(* IEC 61131-3 sources: mect_apps/TPAC1008/RemoteControl_PLC, 7 files *)

(* ---- ImpostazioniCAN1.gvl ---- *)
(* Global var file *)
VAR_GLOBAL
	ch1_CAN1_IN_DIG_8_1 AT %IB3.4096: BYTE;
	ch1_CAN1_IN_DIG_8_2 AT %IB3.4097: BYTE;
	ch1_CAN1_OUT_DIG_8_1 AT %QB3.4096: BYTE;

	ch1_CAN1_OUT_DIG_8_1_7 AT %QX3.4096.7: BOOL;

	ch1_CAN1_OUT_DIG_8_2 AT %QB3.4097: BYTE;
	ch1_CAN1_IN_AN_1 AT %IW3.8192: INT;
	ch1_CAN1_IN_AN_2 AT %IW3.8194: INT;
	ch1_CAN1_IN_AN_3 AT %IW3.8196: INT;
	ch1_CAN1_IN_AN_4 AT %IW3.8198: INT;
	ch1_CAN1_IN_AN_5 AT %IW3.8200: INT;
	ch1_CAN1_IN_AN_6 AT %IW3.8202: INT;
	ch1_CAN1_IN_AN_7 AT %IW3.8204: INT;
	ch1_CAN1_IN_AN_8 AT %IW3.8206: INT;
	ch1_CAN1_IN_AN_9 AT %IW3.8208: INT;
	ch1_CAN1_IN_AN_10 AT %IW3.8210: INT;
	ch1_CAN1_IN_AN_11 AT %IW3.8212: INT;
	ch1_CAN1_IN_AN_12 AT %IW3.8214: INT;
	ch1_CAN1_IN_AN_13 AT %IW3.8216: INT;
	ch1_CAN1_IN_AN_14 AT %IW3.8218: INT;
	ch1_CAN1_IN_AN_15 AT %IW3.8220: INT;
	ch1_CAN1_IN_AN_16 AT %IW3.8222: INT;
	ch1_CAN1_OUT_AN_1 AT %QW3.8192: INT;
	PLC_CAN1_IN_DIG_8_1 AT %MB0.21200: BYTE;

	PLC_CAN1_IN_DIG_8_2 AT %MB0.21204: BYTE;
	PLC_CAN1_OUT_DIG_8_1 AT %MB0.21208: BYTE;
	PLC_CAN1_OUT_DIG_8_1_0 AT %MX0.21208.0: BOOL;
	PLC_CAN1_OUT_DIG_8_1_1 AT %MX0.21208.1: BOOL;
	PLC_CAN1_OUT_DIG_8_1_2 AT %MX0.21208.2: BOOL;
	PLC_CAN1_OUT_DIG_8_1_3 AT %MX0.21208.3: BOOL;
	PLC_CAN1_OUT_DIG_8_1_4 AT %MX0.21208.4: BOOL;
	PLC_CAN1_OUT_DIG_8_1_5 AT %MX0.21208.5: BOOL;
	PLC_CAN1_OUT_DIG_8_1_6 AT %MX0.21208.6: BOOL;
	PLC_CAN1_OUT_DIG_8_1_7 AT %MX0.21208.7: BOOL;

	PLC_CAN1_OUT_DIG_8_2 AT %MB0.21212: BYTE;

	PLC_CAN1_IN_AN_1 AT %MW0.21216: INT;
	PLC_CAN1_IN_AN_2 AT %MW0.21220: INT;
	PLC_CAN1_IN_AN_3 AT %MW0.21224: INT;
	PLC_CAN1_IN_AN_4 AT %MW0.21228: INT;
	PLC_CAN1_IN_AN_5 AT %MW0.21232: INT;
	PLC_CAN1_IN_AN_6 AT %MW0.21236: INT;
	PLC_CAN1_IN_AN_7 AT %MW0.21240: INT;
	PLC_CAN1_IN_AN_8 AT %MW0.21244: INT;
	PLC_CAN1_IN_AN_9 AT %MW0.21248: INT;
	PLC_CAN1_IN_AN_10 AT %MW0.21252: INT;
	PLC_CAN1_IN_AN_11 AT %MW0.21256: INT;
	PLC_CAN1_IN_AN_12 AT %MW0.21260: INT;
	PLC_CAN1_IN_AN_13 AT %MW0.21264: INT;
	PLC_CAN1_IN_AN_14 AT %MW0.21268: INT;
	PLC_CAN1_IN_AN_15 AT %MW0.21272: INT;
	PLC_CAN1_IN_AN_16 AT %MW0.21276: INT;
	PLC_CAN1_OUT_AN_1 AT %MW0.21280: INT;
END_VAR

(* ---- Resource1.gvl ---- *)
(* Global variable file *)
VAR_GLOBAL

	Selection AT %MW0.4:UINT;
	ISI_S1_GRU AT %MW0.8:INT;
	FSI_S1_GRU AT %MW0.12:INT;
	ISL_S1_GRU AT %MW0.16:INT;
	FSL_S1_GRU AT %MW0.20:INT;
	ISI_S2_GRU AT %MW0.24:INT;
	FSI_S2_GRU AT %MW0.28:INT;
	ISL_S2_GRU AT %MW0.32:INT;
	FSL_S2_GRU AT %MW0.36:INT;
	ISI_S3_GRU AT %MW0.40:INT;
	FSI_S3_GRU AT %MW0.44:INT;
	ISL_S3_GRU AT %MW0.48:INT;
	FSL_S3_GRU AT %MW0.52:INT;
	ISI_S1_ESC AT %MW0.56:INT;
	FSI_S1_ESC AT %MW0.60:INT;
	ISL_S1_ESC AT %MW0.64:INT;
	FSL_S1_ESC AT %MW0.68:INT;
	ISI_S2_ESC AT %MW0.72:INT;
	FSI_S2_ESC AT %MW0.76:INT;
	ISL_S2_ESC AT %MW0.80:INT;
	FSL_S2_ESC AT %MW0.84:INT;
	ISI_S3_ESC AT %MW0.88:INT;
	FSI_S3_ESC AT %MW0.92:INT;
	ISL_S3_ESC AT %MW0.96:INT;
	FSL_S3_ESC AT %MW0.100:INT;
	ZERO_S1_GRU AT %MW0.104:INT;
	ZERO_S2_GRU AT %MW0.108:INT;
	ZERO_S3_GRU AT %MW0.112:INT;
	ZERO_S1_ESC AT %MW0.116:INT;
	ZERO_S2_ESC AT %MW0.120:INT;
	ZERO_S3_ESC AT %MW0.124:INT;
	manual AT %MW0.128:UINT;
	DigitalOutput_1 AT %MD0.5380:UDINT;
	DigitalOutput_2 AT %MD0.5384:UDINT;
	DigitalInput_3 AT %MD0.5388:UDINT;
	DigitalInput_4 AT %MD0.5392:UDINT;
	TimeValue AT %MD0.5396:REAL;
	TimeMin AT %MD0.5400:REAL;
	TimeMax AT %MD0.5404:REAL;
	AnalogInput_1 AT %MW0.5408:INT;
	AnalogInput_2 AT %MW0.5412:INT;
	Mesaure_gru1 AT %MW0.5416:INT;
	Mesaure_gru2 AT %MW0.5420:INT;
	Mesaure_gru3 AT %MW0.5424:INT;
	Mesaure_esc1 AT %MW0.5428:INT;
	Mesaure_esc2 AT %MW0.5432:INT;
	Mesaure_esc3 AT %MW0.5436:INT;
	Tasto1 AT %MW0.5440:INT;
	Tasto2 AT %MW0.5444:INT;
	Tasto3 AT %MW0.5448:INT;
	Tasto4 AT %MW0.5452:INT;
	Tasto5 AT %MW0.5456:INT;
	Tasto6 AT %MW0.5460:INT;

	step1T AT %MW0.5464:INT;
	step1M AT %MW0.5468:INT;
	step2T AT %MW0.5472:INT;
	step2M AT %MW0.5476:INT;
	step3T AT %MW0.5480:INT;
	step3M AT %MW0.5484:INT;
	step4T AT %MW0.5488:INT;
	step4M AT %MW0.5492:INT;
	step5T AT %MW0.5496:INT;
	step5M AT %MW0.5500:INT;
	step6T AT %MW0.5504:INT;
	step6M AT %MW0.5508:INT;
	step7T AT %MW0.5512:INT;
	step7M AT %MW0.5516:INT;
	step8T AT %MW0.5520:INT;
	step8M AT %MW0.5524:INT;
	step9T AT %MW0.5528:INT;
	step9M AT %MW0.5532:INT;
	step10T AT %MW0.5536:INT;
	step10M AT %MW0.5540:INT;
	SetZ_gru1 AT %MW0.5544:INT;
	SetZ_gru2 AT %MW0.5548:INT;
	SetZ_gru3 AT %MW0.5552:INT;
	SetZ_esc1 AT %MW0.5556:INT;
	SetZ_esc2 AT %MW0.5560:INT;
	SetZ_esc3 AT %MW0.5564:INT;

	Offset_AnIn_1_GRU:INT;
	Offset_AnIn_2_GRU:INT;
	Offset_AnIn_3_GRU:INT;
	Offset_AnIn_1_ESC:INT;
	Offset_AnIn_2_ESC:INT;
	Offset_AnIn_3_ESC:INT;

END_VAR

(* ---- TPACLocaIO.gvl ---- *)
(*Global variable file*)
(*[[
]]*)
VAR_GLOBAL
	PLC_DigIn_1 AT %MW0.21200:WORD;
	PLC_DigIn_2 AT %MW0.21204:WORD;
	PLC_DigIn_3 AT %MW0.21208:WORD;
	PLC_DigIn_4 AT %MW0.21212:WORD;
	PLC_DigIn_5 AT %MW0.21216:WORD;
	PLC_DigIn_6 AT %MW0.21220:WORD;
	PLC_DigIn_7 AT %MW0.21224:WORD;
	PLC_DigIn_8 AT %MW0.21228:WORD;
	PLC_DigIn_9 AT %MW0.21232:WORD;
	PLC_DigIn_10 AT %MW0.21236:WORD;
	PLC_DigIn_11 AT %MW0.21240:WORD;
	PLC_DigIn_12 AT %MW0.21244:WORD;
	PLC_DigIn_13 AT %MW0.21248:WORD;
	PLC_DigIn_14 AT %MW0.21252:WORD;
	PLC_DigIn_15 AT %MW0.21256:WORD;
	PLC_DigIn_16 AT %MW0.21260:WORD;
	PLC_DigOut_1 AT %MW0.21264:WORD;
	PLC_DigOut_2 AT %MW0.21268:WORD;
	PLC_DigOut_3 AT %MW0.21272:WORD;
	PLC_DigOut_4 AT %MW0.21276:WORD;
	PLC_DigOut_5 AT %MW0.21280:WORD;
	PLC_DigOut_6 AT %MW0.21284:WORD;
	PLC_DigOut_7 AT %MW0.21288:WORD;
	PLC_DigOut_8 AT %MW0.21292:WORD;
	PLC_DigOut_9 AT %MW0.21296:WORD;
	PLC_DigOut_10 AT %MW0.21300:WORD;
	PLC_DigOut_11 AT %MW0.21304:WORD;
	PLC_DigOut_12 AT %MW0.21308:WORD;
	PLC_DigOut_13 AT %MW0.21312:WORD;
	PLC_DigOut_14 AT %MW0.21316:WORD;
	PLC_DigOut_15 AT %MW0.21320:WORD;
	PLC_DigOut_16 AT %MW0.21324:WORD;
	PLC_DigDir_1 AT %MW0.21328:WORD;
	PLC_DigDir_2 AT %MW0.21332:WORD;
	PLC_DigDir_3 AT %MW0.21336:WORD;
	PLC_DigDir_4 AT %MW0.21340:WORD;
	PLC_DigDir_5 AT %MW0.21344:WORD;
	PLC_DigDir_6 AT %MW0.21348:WORD;
	PLC_DigDir_7 AT %MW0.21352:WORD;
	PLC_DigDir_8 AT %MW0.21356:WORD;
	PLC_DigDir_9 AT %MW0.21360:WORD;
	PLC_DigDir_10 AT %MW0.21364:WORD;
	PLC_DigDir_11 AT %MW0.21368:WORD;
	PLC_DigDir_12 AT %MW0.21372:WORD;
	PLC_DigDir_13 AT %MW0.21376:WORD;
	PLC_DigDir_14 AT %MW0.21380:WORD;
	PLC_DigDir_15 AT %MW0.21384:WORD;
	PLC_DigDir_16 AT %MW0.21388:WORD;
	PLC_AnIn_1 AT %MW0.21392:INT;
	PLC_AnIn_2 AT %MW0.21396:INT;
	PLC_AnIn_3 AT %MW0.21400:INT;
	PLC_AnIn_4 AT %MW0.21404:INT;
	PLC_AnIn_5 AT %MW0.21408:INT;
	PLC_AnIn_6 AT %MW0.21412:INT;
	PLC_AnIn_7 AT %MW0.21416:INT;
	PLC_AnIn_8 AT %MW0.21420:INT;
	PLC_AnOut_1  AT %MW0.21424:INT;
	PLC_AnOut_2 AT %MW0.21428:INT;
	PLC_AnOut_3  AT %MW0.21432:INT;
	PLC_AnOut_4 AT %MW0.21436:INT;
	PLC_AnOut_5  AT %MW0.21440:INT;
	PLC_AnOut_6 AT %MW0.21444:INT;
	PLC_AnOut_7  AT %MW0.21448:INT;
	PLC_AnOut_8 AT %MW0.21452:INT;
	PLC_AnInConf_1 AT %MW0.21456:WORD;
	PLC_AnInConf_2 AT %MW0.21460:WORD;
	PLC_AnInConf_3 AT %MW0.21464:WORD;
	PLC_AnInConf_4 AT %MW0.21468:WORD;
	PLC_AnInConf_5 AT %MW0.21472:WORD;
	PLC_AnInConf_6 AT %MW0.21476:WORD;
	PLC_AnInConf_7 AT %MW0.21480:WORD;
	PLC_AnInConf_8 AT %MW0.21484:WORD;
	PLC_AnOutConf_1 AT %MW0.21488:WORD;
	PLC_AnOutConf_2 AT %MW0.21492:WORD;
	PLC_AnOutConf_3 AT %MW0.21496:WORD;
	PLC_AnOutConf_4 AT %MW0.21500:WORD;
	PLC_AnOutConf_5 AT %MW0.21504:WORD;
	PLC_AnOutConf_6 AT %MW0.21508:WORD;
	PLC_AnOutConf_7 AT %MW0.21512:WORD;
	PLC_AnOutConf_8 AT %MW0.21516:WORD;
	PLC_Tamb AT %MW0.21520:INT;
	PLC_EncoderLo AT %MW0.21524:UINT;
	PLC_EncoderHi AT %MW0.21528:UINT;
	PLC_StatusReg AT %MW0.21532:UINT;
	PLC_ControlWord  AT %MW0.21536:WORD;
	PLC_EncoderPreset_Lo AT %MW0.21540:UINT;
	PLC_EncoderPreset_Hi AT %MW0.21544:UINT;
	PLC_EncoderReset AT %MW0.21548:WORD;
	PLC_EncoderEnable AT %MW0.21552:WORD;
	PLC_RPM AT %MW0.21556:UINT;
	PLC_time AT %MD0.21560:REAL;
	PLC_timeMin AT %MD0.21564:REAL;
	PLC_timeMax AT %MD0.21568:REAL;
END_VAR

(* ---- fb_TPAC1006_LIOsync.st ---- *)
(*[[
]]*)
FUNCTION_BLOCK fb_TPAC1006_LIOsync
#import "LIO_TPAC1006.gvl"
#import "TPACLocaIO.gvl"
#import "crosstable.gvl"
VAR_INPUT
END_VAR
VAR
END_VAR
IF (HardwareType AND 16#000000FF) >= 16#1 THEN
	IF (UINT_TO_WORD(TP1006_LIO_StatusReg) AND 16#01) = 1 	 THEN

		PLC_DigIn_1:=BOOL_TO_WORD(TP1006_LIO_DigIn_1);
		PLC_DigIn_2:=BOOL_TO_WORD(TP1006_LIO_DigIn_2);
		PLC_DigIn_3:=BOOL_TO_WORD(TP1006_LIO_DigIn_3);
		PLC_DigIn_4:=BOOL_TO_WORD(TP1006_LIO_DigIn_4);
		PLC_DigIn_5:=BOOL_TO_WORD(TP1006_LIO_DigIn_5);
		PLC_DigIn_6:=BOOL_TO_WORD(TP1006_LIO_DigIn_6);
		PLC_DigIn_7:=BOOL_TO_WORD(TP1006_LIO_DigIn_7);
		PLC_DigIn_8:=BOOL_TO_WORD(TP1006_LIO_DigIn_8);

		PLC_DigIn_9:=BOOL_TO_WORD(TP1006_LIO_DigIn_9);
		PLC_DigIn_10:=BOOL_TO_WORD(TP1006_LIO_DigIn_10);
		PLC_DigIn_11:=BOOL_TO_WORD(TP1006_LIO_DigIn_11);
		PLC_DigIn_12:=BOOL_TO_WORD(TP1006_LIO_DigIn_12);
		PLC_DigIn_13:=BOOL_TO_WORD(TP1006_LIO_DigIn_13);
		PLC_DigIn_14:=BOOL_TO_WORD(TP1006_LIO_DigIn_14);
		PLC_DigIn_15:=BOOL_TO_WORD(TP1006_LIO_DigIn_15);
		PLC_DigIn_16:=BOOL_TO_WORD(TP1006_LIO_DigIn_16);

		TP1006_LIO_DigOut_1:=WORD_TO_BOOL(PLC_DigOut_1);
		TP1006_LIO_DigOut_2:=WORD_TO_BOOL(PLC_DigOut_2);
		TP1006_LIO_DigOut_3:=WORD_TO_BOOL(PLC_DigOut_3);
		TP1006_LIO_DigOut_4:=WORD_TO_BOOL(PLC_DigOut_4);
		TP1006_LIO_DigOut_5:=WORD_TO_BOOL(PLC_DigOut_5);
		TP1006_LIO_DigOut_6:=WORD_TO_BOOL(PLC_DigOut_6);
		TP1006_LIO_DigOut_7:=WORD_TO_BOOL(PLC_DigOut_7);
		TP1006_LIO_DigOut_8:=WORD_TO_BOOL(PLC_DigOut_8);

		TP1006_LIO_DigOut_9:=WORD_TO_BOOL(PLC_DigOut_9);
		TP1006_LIO_DigOut_10:=WORD_TO_BOOL(PLC_DigOut_10);
		TP1006_LIO_DigOut_11:=WORD_TO_BOOL(PLC_DigOut_11);
		TP1006_LIO_DigOut_12:=WORD_TO_BOOL(PLC_DigOut_12);
		TP1006_LIO_DigOut_13:=WORD_TO_BOOL(PLC_DigOut_13);
		TP1006_LIO_DigOut_14:=WORD_TO_BOOL(PLC_DigOut_14);
		TP1006_LIO_DigOut_15:=WORD_TO_BOOL(PLC_DigOut_15);
		TP1006_LIO_DigOut_16:=WORD_TO_BOOL(PLC_DigOut_16);

		PLC_AnIn_1:= TP1006_LIO_AnIn_1;
		PLC_AnIn_2:= TP1006_LIO_AnIn_2;
		PLC_AnIn_3:= TP1006_LIO_AnIn_3;
		PLC_AnIn_4:= TP1006_LIO_AnIn_4;

		PLC_Tamb:= TP1006_LIO_Tamb;
		PLC_EncoderLo:= TP1006_LIO_EncoderLo;
		PLC_EncoderHi:= TP1006_LIO_EncoderHi;
		PLC_StatusReg:= TP1006_LIO_StatusReg;
		PLC_RPM:= TP1006_LIO_RPM;
		TP1006_LIO_AnIn_Conf:=WORD_TO_INT(PLC_AnInConf_1 OR SHL(PLC_AnInConf_2,4) OR SHL(PLC_AnInConf_3,8) OR SHL(PLC_AnInConf_4,12) );
		TP1006_LIO_AnOut_Conf:=WORD_TO_INT(INT_TO_WORD(WORD_TO_INT(PLC_AnOutConf_1)) OR SHL(INT_TO_WORD(WORD_TO_INT(PLC_AnOutConf_2)),4) );

		TP1006_LIO_AnOut_1:= PLC_AnOut_1;
		TP1006_LIO_AnOut_2:= PLC_AnOut_2;
		TP1006_LIO_ControlWord:= PLC_ControlWord;
		TP1006_LIO_EncoderPreset_Lo:= PLC_EncoderPreset_Lo;
		TP1006_LIO_EncoderPreset_hI:= PLC_EncoderPreset_Hi;
	END_IF;

END_IF;

END_FUNCTION_BLOCK

(* ---- fb_TPAC1007_LIOsync.st ---- *)
(*[[
]]*)
FUNCTION_BLOCK fb_TPAC1007_LIOsync
#import "LIO_TPAC1007.gvl"
#import "TPACLocaIO.gvl"
#import "crosstable.gvl"
VAR_INPUT
END_VAR
VAR
	tmp_dig_out: BYTE;
	tmp_dig_outold:BYTE;
	tmp_dig_dir: BYTE;
	tmp_dig_dirold:BYTE;
END_VAR

IF (HardwareType AND 16#00FF0000) >= 16#1 THEN
		PLC_StatusReg:=TP1007_LIO_Revision;
		PLC_DigIn_1:=BOOL_TO_WORD(TP1007_LIO_DigIn_1);
		PLC_DigIn_2:=BOOL_TO_WORD(TP1007_LIO_DigIn_2);
		PLC_DigIn_3:=BOOL_TO_WORD(TP1007_LIO_DigIn_3);
		PLC_DigIn_4:=BOOL_TO_WORD(TP1007_LIO_DigIn_4);
		PLC_DigIn_5:=BOOL_TO_WORD(TP1007_LIO_DigIn_5);
		PLC_DigIn_6:=BOOL_TO_WORD(TP1007_LIO_DigIn_6);
		PLC_DigIn_7:=BOOL_TO_WORD(TP1007_LIO_DigIn_7);
		PLC_DigIn_8:=BOOL_TO_WORD(TP1007_LIO_DigIn_8);
		PLC_DigIn_9:=BOOL_TO_WORD(TP1007_LIO_DigIn_9);
		PLC_DigIn_10:=BOOL_TO_WORD(TP1007_LIO_DigIn_10);
		PLC_DigIn_11:=BOOL_TO_WORD(TP1007_LIO_DigIn_11);
		PLC_DigIn_12:=BOOL_TO_WORD(TP1007_LIO_DigIn_12);

		PLC_Tamb:= TP1007_LIO_Tamb;
		PLC_EncoderLo:= TP1007_LIO_EncoderLo;
		PLC_EncoderHi:= TP1007_LIO_EncoderHi;

		PLC_AnIn_1 := TP1007_LIO_AnIn_1;
		PLC_AnIn_2 := TP1007_LIO_AnIn_2;

(*SCRITTURA 1*)
		tmp_dig_dir := WORD_TO_BYTE(PLC_DigDir_1 OR SHL(PLC_DigDir_2,1) OR SHL(PLC_DigDir_3,2) OR SHL(PLC_DigDir_4,3) OR SHL(PLC_DigDir_5,4) OR SHL(PLC_DigDir_6,5) OR SHL(PLC_DigDir_7,6) OR SHL(PLC_DigDir_8,7) );
		IF tmp_dig_dir <> tmp_dig_dirold THEN
			TP1007_LIO_DigDir_1_8 := tmp_dig_dir;
		END_IF;
		tmp_dig_dirold := tmp_dig_dir;

(*SCRITTURA 2*)
		tmp_dig_out:= WORD_TO_BYTE(PLC_DigOut_1 OR SHL(PLC_DigOut_2,1) OR SHL(PLC_DigOut_3,2) OR SHL(PLC_DigOut_4,3) OR SHL(PLC_DigOut_5,4) OR SHL(PLC_DigOut_6,5) OR SHL(PLC_DigOut_7,6) OR SHL(PLC_DigOut_8,7) );
		IF tmp_dig_out<> tmp_dig_outold THEN
			TP1007_LIO_DigOut_1_8:= tmp_dig_out;
		END_IF;
		tmp_dig_outold:=tmp_dig_out;

(*SCRITTURA 3*)
		IF PLC_AnInConf_1 <> TP1007_LIO_AnInConf_1 THEN
			TP1007_LIO_AnInConf_1 := PLC_AnInConf_1 ;
		END_IF;
(*SCRITTURA 4*)
		IF PLC_AnInConf_2 <> TP1007_LIO_AnInConf_2 THEN
			TP1007_LIO_AnInConf_2 := PLC_AnInConf_2 ;
		END_IF;
(*SCRITTURA 5*)
		IF PLC_AnOutConf_1 <> TP1007_LIO_AnOut_Conf THEN
			TP1007_LIO_AnOut_Conf := PLC_AnOutConf_1;
		END_IF;
(*SCRITTURA 6*)
		IF PLC_AnOut_1 <> (TP1007_LIO_AnOut_1) THEN
			TP1007_LIO_AnOut_1 := PLC_AnOut_1;
		END_IF;
(*SCRITTURA 7*)
		IF PLC_EncoderReset <> TP1007_LIO_EncoderReset THEN
			TP1007_LIO_EncoderReset := PLC_EncoderReset;
		END_IF;
(*SCRITTURA 8*)
		IF PLC_EncoderEnable <> TP1007_LIO_EncoderEnable THEN
			TP1007_LIO_EncoderEnable := PLC_EncoderEnable;
		END_IF;

END_IF;
END_FUNCTION_BLOCK

(* ---- PLC.st ---- *)
(*[[
]]*)
PROGRAM PLC
#import "crosstable.gvl"
#import "Resource1.gvl"
#import "LIO_TPAC1006.gvl"
#import "TPACLocaIO.gvl"
VAR
	FIRST_CYCLE:BOOL;
	LAST_BUTTON :UINT;
	TMP1:REAL;
	TMP2:REAL;
END_VAR;
	IF NOT FIRST_CYCLE THEN
		IF Selection > 0 THEN
(*
			ISI_S1_GRU:=4000;
			FSI_S1_GRU:=20000;
			ISI_S2_GRU:=4000;
			FSI_S2_GRU:=20000;
			ISI_S3_GRU:=4000;
			FSI_S3_GRU:=20000;
			ISI_S1_ESC:=4000;
			FSI_S1_ESC:=20000;
			ISI_S2_ESC:=4000;
			FSI_S2_ESC:=20000;
			ISI_S3_ESC:=4000;
			FSI_S3_ESC:=20000;

			ISL_S1_GRU:=0;
			FSL_S1_GRU:=3600;
			ISL_S2_GRU:=0;
			FSL_S2_GRU:=3600;
			ISL_S3_GRU:=-900;
			FSL_S3_GRU:=900;
			ISL_S1_ESC:=0;
			FSL_S1_ESC:=3000;
			ISL_S2_ESC:=0;
			FSL_S2_ESC:=3600;
			ISL_S3_ESC:=-900;
			FSL_S3_ESC:=900;
	*)
			FIRST_CYCLE:=TRUE;
		END_IF;
	ELSE
		IF Selection =1 THEN
			PLC_AnInConf_1:=1;
			PLC_AnInConf_2:=1;
			PLC_AnInConf_3:=2;
			PLC_AnInConf_4:=0;
		ELSE
			PLC_AnInConf_1:=1;
			PLC_AnInConf_2:=1;
			PLC_AnInConf_3:=1;
			PLC_AnInConf_4:=0;
		END_IF;
		IF SetZ_gru1 =1 THEN
			ZERO_S1_GRU:=PLC_AnIn_1;
		END_IF;

		IF SetZ_gru2 = 1 THEN
			ZERO_S2_GRU:=PLC_AnIn_2;
		END_IF;

		IF SetZ_gru3 = 1 THEN
			ZERO_S3_GRU:=PLC_AnIn_3;
		END_IF;

		IF SetZ_esc1  = 1 THEN
			ZERO_S1_ESC:=PLC_AnIn_1;
		END_IF;

		IF SetZ_esc2  = 1 THEN
			ZERO_S2_ESC:=PLC_AnIn_2;
		END_IF;

		IF SetZ_esc3  = 1 THEN
			ZERO_S3_ESC:=PLC_AnIn_3;
		END_IF;

		IF Selection = 2 THEN
			IF Tasto1 =1 THEN
				IF LAST_BUTTON <> 1 THEN
					PLC_DigOut_1:=0;
					PLC_DigOut_2:=0;
					LAST_BUTTON:=1;
				ELSE
					PLC_DigOut_1:=1;
					PLC_DigOut_2:=0;
					PLC_DigOut_3:=0;
				END_IF;
			ELSIF Tasto2 =1 THEN
				IF LAST_BUTTON <> 2 THEN
					PLC_DigOut_1:=0;
					PLC_DigOut_2:=0;
					LAST_BUTTON:=2;
				ELSE
					PLC_DigOut_1:=0;
					PLC_DigOut_2:=1;
					PLC_DigOut_3:=1;
				END_IF;
			ELSIF Tasto3 =1 THEN
				IF LAST_BUTTON <> 3 THEN
					PLC_DigOut_4:=0;
					PLC_DigOut_5:=0;
					LAST_BUTTON:=3;
				ELSE
					PLC_DigOut_4:=1;
					PLC_DigOut_5:=0;
					PLC_DigOut_6:=0;
				END_IF;
			ELSIF Tasto4 =1 THEN
				IF LAST_BUTTON <> 4 THEN
					PLC_DigOut_4:=0;
					PLC_DigOut_5:=0;
					LAST_BUTTON:=4;
				ELSE
					PLC_DigOut_4:=0;
					PLC_DigOut_5:=1;
					PLC_DigOut_6:=1;
				END_IF;
			ELSIF Tasto5 =1 THEN
				IF LAST_BUTTON <> 5 THEN
					PLC_DigOut_7:=0;
					PLC_DigOut_8:=0;
					LAST_BUTTON:=5;
				ELSE
					PLC_DigOut_7:=1;
					PLC_DigOut_8:=0;
					PLC_DigOut_9:=0;
				END_IF;
			ELSIF Tasto6 =1 THEN
				IF LAST_BUTTON <> 6 THEN
					PLC_DigOut_7:=0;
					PLC_DigOut_8:=0;
					LAST_BUTTON:=6;
				ELSE
					PLC_DigOut_7:=0;
					PLC_DigOut_8:=1;
					PLC_DigOut_9:=1;
				END_IF;
			ELSIF Tasto1=0 AND Tasto2=0 AND Tasto3=0 AND Tasto4=0 AND Tasto5=0 AND Tasto6=0 THEN
				PLC_DigOut_1:=0;
				PLC_DigOut_2:=0;
				PLC_DigOut_4:=0;
				PLC_DigOut_5:=0;
				PLC_DigOut_7:=0;
				PLC_DigOut_8:=0;
			END_IF;

			IF(FSI_S1_ESC-ISI_S1_ESC) > 0 THEN
				TMP1:=INT_TO_REAL((ZERO_S1_ESC-ISI_S1_ESC))*int_to_real((FSL_S1_ESC-ISL_S1_ESC))/INT_TO_REAL((FSI_S1_ESC-ISI_S1_ESC))+INT_TO_REAL(ISL_S1_ESC);
				TMP2:=INT_TO_REAL((PLC_AnIn_1-ISI_S1_ESC))*int_to_real((FSL_S1_ESC-ISL_S1_ESC))/INT_TO_REAL((FSI_S1_ESC-ISI_S1_ESC))+INT_TO_REAL(ISL_S1_ESC);
				Mesaure_ESC1:=REAL_TO_INT(TMP2-TMP1);
			END_IF;
			IF(FSI_S2_ESC-ISI_S2_ESC) > 0 THEN
				TMP1:=INT_TO_REAL((ZERO_S2_ESC-ISI_S2_ESC))*int_to_real((FSL_S2_ESC-ISL_S2_ESC))/INT_TO_REAL((FSI_S2_ESC-ISI_S2_ESC))+INT_TO_REAL(ISL_S2_ESC);
				TMP2:=INT_TO_REAL((PLC_AnIn_2-ISI_S2_ESC))*int_to_real((FSL_S2_ESC-ISL_S2_ESC))/INT_TO_REAL((FSI_S2_ESC-ISI_S2_ESC))+INT_TO_REAL(ISL_S2_ESC);
				Mesaure_ESC2:=REAL_TO_INT(TMP2-TMP1);
			END_IF;
			IF(FSI_S3_ESC-ISI_S3_ESC) > 0 THEN
				TMP1:=INT_TO_REAL((ZERO_S3_ESC-ISI_S3_ESC))*int_to_real((FSL_S3_ESC-ISL_S3_ESC))/INT_TO_REAL((FSI_S3_ESC-ISI_S3_ESC))+INT_TO_REAL(ISL_S3_ESC);
				TMP2:=INT_TO_REAL((PLC_AnIn_3-ISI_S3_ESC))*int_to_real((FSL_S3_ESC-ISL_S3_ESC))/INT_TO_REAL((FSI_S3_ESC-ISI_S3_ESC))+INT_TO_REAL(ISL_S3_ESC);
				Mesaure_ESC3:=REAL_TO_INT(TMP2-TMP1);

			END_IF;

		ELSIF Selection = 1 THEN
			IF Tasto1 =1 THEN
				IF LAST_BUTTON <> 1 THEN
					PLC_DigOut_1:=0;
					PLC_DigOut_2:=0;
					LAST_BUTTON:=1;
				ELSE
					PLC_DigOut_1:=1;
					PLC_DigOut_2:=0;
				END_IF;
			ELSIF Tasto2 =1 THEN
				IF LAST_BUTTON <> 2 THEN
					PLC_DigOut_1:=0;
					PLC_DigOut_2:=0;
					LAST_BUTTON:=2;
				ELSE
					PLC_DigOut_1:=0;
					PLC_DigOut_2:=1;
				END_IF;
			ELSIF Tasto3 =1 THEN
				IF LAST_BUTTON <> 3 THEN
					PLC_DigOut_3:=0;
					PLC_DigOut_4:=0;
					LAST_BUTTON:=3;
				ELSE
					PLC_DigOut_3:=1;
					PLC_DigOut_4:=0;
				END_IF;
			ELSIF Tasto4 =1 THEN
				IF LAST_BUTTON <> 4 THEN
					PLC_DigOut_3:=0;
					PLC_DigOut_4:=0;
					LAST_BUTTON:=4;
				ELSE
					PLC_DigOut_3:=0;
					PLC_DigOut_4:=1;
				END_IF;
			ELSIF Tasto1=0 AND Tasto2=0 AND Tasto3=0 AND Tasto4=0 AND Tasto5=0 AND Tasto6=0 THEN
				PLC_DigOut_1:=0;
				PLC_DigOut_2:=0;
				PLC_DigOut_3:=0;
				PLC_DigOut_4:=0;
				PLC_DigOut_7:=0;
				PLC_DigOut_8:=0;
			END_IF;

			IF(FSI_S1_GRU-ISI_S1_GRU) > 0 THEN
				TMP1:=INT_TO_REAL((ZERO_S1_GRU-ISI_S1_GRU))*int_to_real((FSL_S1_GRU-ISL_S1_GRU))/INT_TO_REAL((FSI_S1_GRU-ISI_S1_GRU))+INT_TO_REAL(ISL_S1_GRU);
				TMP2:=INT_TO_REAL((PLC_AnIn_1-ISI_S1_GRU))*int_to_real((FSL_S1_GRU-ISL_S1_GRU))/INT_TO_REAL((FSI_S1_GRU-ISI_S1_GRU))+INT_TO_REAL(ISL_S1_GRU);
				Mesaure_gru1:=REAL_TO_INT(TMP2-TMP1);
			END_IF;
			IF(FSI_S2_GRU-ISI_S2_GRU) > 0 THEN
				TMP1:=INT_TO_REAL((ZERO_S2_GRU-ISI_S2_GRU))*int_to_real((FSL_S2_GRU-ISL_S2_GRU))/INT_TO_REAL((FSI_S2_GRU-ISI_S2_GRU))+INT_TO_REAL(ISL_S2_GRU);
				TMP2:=INT_TO_REAL((PLC_AnIn_2-ISI_S2_GRU))*int_to_real((FSL_S2_GRU-ISL_S2_GRU))/INT_TO_REAL((FSI_S2_GRU-ISI_S2_GRU))+INT_TO_REAL(ISL_S2_GRU);
				Mesaure_gru2:=REAL_TO_INT(TMP2-TMP1);
			END_IF;
			IF(FSI_S3_GRU-ISI_S3_GRU) > 0 THEN
				TMP1:=INT_TO_REAL((ZERO_S3_GRU-ISI_S3_GRU))*int_to_real((FSL_S3_GRU-ISL_S3_GRU))/INT_TO_REAL((FSI_S3_GRU-ISI_S3_GRU))+INT_TO_REAL(ISL_S3_GRU);
				TMP2:=INT_TO_REAL((PLC_AnIn_3-ISI_S3_GRU))*int_to_real((FSL_S3_GRU-ISL_S3_GRU))/INT_TO_REAL((FSI_S3_GRU-ISI_S3_GRU))+INT_TO_REAL(ISL_S3_GRU);
				Mesaure_gru3:=REAL_TO_INT(TMP2-TMP1);
			END_IF;

		END_IF;
		IF manual = 0 THEN
			IF Selection=1 THEN

		;

			ELSIF Selection=2 THEN

		;

			END_IF;

		END_IF;
	END_IF;
END_PROGRAM

(* ---- TCPRTU_Communication.st ---- *)
(*[[
]]*)
PROGRAM TCPRTU_Communication
#import "Resource1.gvl"
#import "crosstable.gvl"

VAR
	HeadAddr:INT;
	ReadWrite:WORD;
	IndexProt_i:ARRAY [0..4] OF INT;
	TON_0:TON;
	TON_1:TON;
	TON_2:TON;
	TON_3:TON;
	BusAccess:fb_HW119_MODBUS;
	FirstCy:BOOL;
	dummy:WORD;
	Enablei: ARRAY [0..3] OF BOOL;
	pointer:INT;
	FlagPrimoCiclo:BOOL;
	Retry:BOOL:=FALSE;
	Protocollo:UINT:=TCPRTU;
	time2:TIME;
	zero:TIME;
	RicettaON:BOOL;
	LastID:INT;
	FirstID:INT;
	I:INT;
	Start:ARRAY [0..4] OF BOOL;
	k:dword;
	j:dword;
END_VAR

TON_0(IN := TRUE,PT := INT_TO_TIME(CommParameters[Protocollo+1].Tmin));
				TON_1(IN := TRUE,PT := DINT_TO_TIME(Talta));
				TON_2(IN := TRUE,PT := DINT_TO_TIME(Tmedia));
				TON_3(IN := TRUE,PT := DINT_TO_TIME(Tbassa));

IF NOT FirstCy THEN
	dummy:=	WD_Disable('Task4_TCPRTU');
	FirstCy:=TRUE;
END_IF;

IF 	TON_0.Q THEN																(* controlla se TIMER Tmin scaduto	*)
	TRIGGER02:=1;
	TRIGGER01:=1;

	TON_0(In:=FALSE);

	IF Reset_TCPRTU =1 THEN
		FOR I:=1 TO 64 DO
			CounterTCPRTU[I]:=0;
		 END_FOR;
		TCPRTUBlackList_ERROR_WORD:=0;
		TCPRTUComm_ERROR_WORD:=0;
		BlackListTCPRTUL:=0;
		BlackListTCPRTUH:=0;
		CommErrTCPRTUL:=0;
		CommErrTCPRTUH:=0;
		ERROR_FLAG:=ERROR_FLAG AND 16#FFFB;

	END_IF;
	IF NOT Retry THEN
		IF TCPRTURequestPLCWrite > 0 THEN											(* controlla seci sono richieste di scrittura da parte del PLC	*)
			pointer:=4;
			FlagPrimoCiclo:=FALSE;
			IndexProt_i[pointer]:=0;
			HeadAddr:=WORD_TO_INT(LocalRTUQueue[IndexRTUQueueGet]);		(*inizializza i parametri da assegnare al blocco funzione*)
			IF CrossTable[HeadAddr].Counter=1 THEN
				ReadWrite:=WRITE_SINGLE;											(*inizializza i parametri da assegnare al blocco funzione*)
			ELSE
				ReadWrite:=WRITE_MULTIPLE;											(*inizializza i parametri da assegnare al blocco funzione*)
			END_IF;
			TCPRTURequestPLCWrite:=TCPRTURequestPLCWrite-1;							(* incrementa il contatore delle scritture effettuate*)
			IndexTCPRTUQueueGet:=IndexTCPRTUQueueGet+1;								(* incrementa il puntatore alla coda *)
			IF IndexTCPRTUQueueGet > MaxLocalQueue THEN
				IndexTCPRTUQueueGet:=0;
			END_IF;
		ELSE
			IF RichiestaScrittura=1 THEN										(* controlla se ci sono richieste di SCRITTURA da parte HMI*)
				IF FlagPrimoCiclo = FALSE THEN									(* controlla se è il primo ingrsso nel ramo a seguito dell'interrupt*)
					FlagPrimoCiclo:=TRUE;										(* Prima richiesta di scrittura => azzero l'indice della coda 	*)
					IndexProt_i[3]:=0;											(* per eseguire le scritture nella sequenza di arrivo		  	*)
					pointer:=3;
					zero:=TIM_Get();
				END_IF;
				REPEAT 															(* Rileva la succssiva variabile a cui accedere nella coda			*)
					IF IndexProt_i[3] < DINT_TO_INT(DimCrossTable) THEN
						IndexProt_i[3]:=IndexProt_i[3]+1;
						ReadWrite:=ARRAY_QUEUE[IndexProt_i[3]] AND QueueRWMask;
						HeadAddr:=WORD_TO_INT(ARRAY_QUEUE[IndexProt_i[3]] AND QueueAddressMask);
						IF HeadAddr < DINT_TO_INT(DimCrossTable) 	THEN
							IF  (ReadWrite = 0  ) OR ( (CrossTable[HeadAddr].Protocol = Protocollo) AND ReadWrite>=WRITE AND (ARRAY_QUEUE_OUTPUT[IndexProt_i[3]]<>STATO_BUSY_WRITE) )   THEN

								IF ReadWrite = 0 THEN
									ARRAY_QUEUE_OUTPUT[IndexProt_i[3]]:=0;
									IF HeadAddr = 0 THEN
										IndexProt_i[3]:=0;
									END_IF;
								ELSIF ReadWrite = WRITE_RIC_SINGLE  OR ReadWrite = WRITE_RIC_MULTIPLE  THEN
									IF NOT RicettaON THEN
										FirstID:=IndexProt_i[3];
										RicettaON:=TRUE;
									END_IF;

									LastID:=IndexProt_i[3];
								END_IF;
								IF ReadWrite>=WRITE THEN
									time2:=TIM_Get()-zero;
								END_IF;

								EXIT;
							END_IF;
						END_IF;
					ELSE
						IndexProt_i[3]:=0;
					END_IF;
				UNTIL  FALSE
				END_REPEAT;
			ELSIF RicettaON AND RichiestaScrittura=0 THEN
				RicettaON:=FALSE;
				FlagPrimoCiclo:=FALSE;
				FOR I:=1 TO  LastID DO
 					ARRAY_QUEUE_OUTPUT[I]:=0;
				END_FOR;
			ELSE																(* richieste di LETTURE	*)
				IF  RichiestaScrittura=0	THEN

					FlagPrimoCiclo:=FALSE;											(* azzera l'akwnoledge dell'interrupt*)
				END_IF;
			END_IF;
			IF  RichiestaScrittura=0	THEN
				IF TON_1.Q OR Enablei[0]=TRUE THEN							(* scaduto il timer ad alta priorità esegue le letture *)
					IF Enablei[0]=FALSE THEN
						TON_1(IN := FALSE);										(* riarma il timer*)
						Start[0]:=TRUE;
					END_IF;
					pointer:=0;
					Enablei[0]:=TRUE;
				ELSIF TON_2.Q OR Enablei[1]=TRUE THEN						(* scaduto il timer ad media priorità esegue le letture *)
					IF Enablei[1]=FALSE THEN
						TON_2(IN := FALSE);										(* riarma il timer*)
						Start[1]:=TRUE;
					END_IF;
					TON_2(IN := FALSE);										(* riarma il timer*)
					pointer:=1;
					Enablei[1]:=TRUE;
				ELSIF TON_3.Q OR Enablei[2]=TRUE THEN						(* scaduto il timer ad media priorità esegue le letture *)
					IF Enablei[2]=FALSE THEN
						TON_3(IN := FALSE);										(* riarma il timer*)
						Start[2]:=TRUE;
					END_IF;
					pointer:=2;
					Enablei[2]:=TRUE;
				END_IF;
		(*		pointer:=0;		*)
				IF Enablei[0] OR Enablei[1] OR Enablei[2] THEN
					REPEAT 															(* Rileva la prima variabile da leggere della cross table*)
						IF IndexProt_i[pointer] < DINT_TO_INT(DimCrossTable) THEN
							IndexProt_i[pointer]:=IndexProt_i[pointer]+1;
							ReadWrite:=ARRAY_QUEUE[IndexProt_i[pointer]] AND QueueRWMask;
							HeadAddr:=WORD_TO_INT(ARRAY_QUEUE[IndexProt_i[pointer]] AND QueueAddressMask);
							IF HeadAddr < DINT_TO_INT(DimCrossTable) 	THEN
								IF ((ReadWrite = 0) OR (CrossTable[HeadAddr].Protocol = Protocollo) AND (CrossTable[HeadAddr].Enable = pointer+1) )    THEN
									IF ReadWrite = 0 THEN
										Enablei[pointer]:=FALSE;
										ARRAY_QUEUE_OUTPUT[IndexProt_i[pointer]]:=0;
										IF HeadAddr = 0 THEN
											IndexProt_i[pointer]:=0;
										END_IF;
									END_IF;
									EXIT;
								END_IF;
							END_IF;
						ELSE
							IndexProt_i[pointer]:=0;
						END_IF;
					UNTIL  FALSE
					END_REPEAT;
				ELSE
					ReadWrite:=0;
				END_IF;

			END_IF;
		END_IF;
	END_IF;
	IF ReadWrite > 0 THEN
		IF Crosstable[HeadAddr].NodeId > 0 AND Crosstable[HeadAddr].NodeId < 64 THEN

			IF TCPRTUListDevices[BYTE_TO_INT(Crosstable[HeadAddr].NodeId)].BlackListed < 2  THEN			(* controlla se il device non è in blacklist*)

				BusAccess(Protocol:='TCPRTU',Index:=IndexProt_i[pointer],address:=HeadAddr,RdWr:=ReadWrite);		(* effettua l'accesso al bus*)
				TON_0(IN := TRUE,PT := INT_TO_TIME(CommParameters[Protocollo+1].Tmin));						(* riarmo di Tmin*)
				IF BusAccess.Error > 0  THEN																(* controlla sec'è stato un errore di comuicazione*)
					ERROR_FLAG:=ERROR_FLAG OR 16#4;
					CounterTCPRTU[BYTE_TO_INT(Crosstable[HeadAddr].NodeId)]:=UDINT_TO_WORD(WORD_TO_UDINT(CounterTCPRTU[BYTE_TO_INT(Crosstable[HeadAddr].NodeId)])+1);
					IF BusAccess.Error = CommError THEN
						TCPRTUComm_ERROR_WORD:=1;
						IF BYTE_TO_INT(Crosstable[HeadAddr].NodeId) > 32 THEN
							CommErrTCPRTUH:=CommErrTCPRTUH OR SHL(16#1,BYTE_TO_INT(Crosstable[HeadAddr].NodeId) -33);
						ELSE
							CommErrTCPRTUL:=CommErrTCPRTUL OR SHL(16#1,BYTE_TO_INT(Crosstable[HeadAddr].NodeId)-1 );
						END_IF;
						Retry:=FALSE;
					ELSIF BusAccess.Error = TimeoutError  THEN		(* controlla se c'è stato un erore di timeout*)
						Retry:=TRUE;							(* imposta il flag retry a TRUE in modo da effettuare le ripetizioni *)
						TCPRTUListDevices[BYTE_TO_INT(Crosstable[HeadAddr].NodeId)].RetryCounter:=TCPRTUListDevices[BYTE_TO_INT(Crosstable[HeadAddr].NodeId)].RetryCounter+1;
						IF TCPRTUListDevices[BYTE_TO_INT(Crosstable[HeadAddr].NodeId)].RetryCounter >= NumberOfFails THEN
							TCPRTUListDevices[BYTE_TO_INT(Crosstable[HeadAddr].NodeId)].BlackListed:=TCPRTUListDevices[BYTE_TO_INT(Crosstable[HeadAddr].NodeId)].BlackListed+1;
							TCPRTUListDevices[BYTE_TO_INT(Crosstable[HeadAddr].NodeId)].JumpRead:=BYTE_TO_INT(FailDivisor);
							Retry:=FALSE;
							IF TCPRTUListDevices[BYTE_TO_INT(Crosstable[HeadAddr].NodeId)].BlackListed > 1 THEN
								TCPRTUBlackList_ERROR_WORD:=1;
								TCPRTU_RUN:=FALSE;
								IF BYTE_TO_INT(Crosstable[HeadAddr].NodeId) > 32 THEN
									BlackListTCPRTUH:=BlackListTCPRTUH OR SHL(16#1,BYTE_TO_INT(Crosstable[HeadAddr].NodeId) -33);
								ELSE
									k:=SHL(16#1,BYTE_TO_INT(Crosstable[HeadAddr].NodeId)-1 );
									BlackListTCPRTUL:=BlackListTCPRTUL OR k;
								END_IF;
							END_IF;
						END_IF;
					END_IF;
				ELSE

					Retry:=FALSE;
					IF BYTE_TO_INT(Crosstable[HeadAddr].NodeId) > 32 THEN
						CommErrTCPRTUH:=CommErrTCPRTUH AND ROL(16#FFFFFFFE,BYTE_TO_INT(Crosstable[HeadAddr].NodeId) -33);
						BlackListTCPRTUH:=BlackListTCPRTUH AND ROL(16#FFFFFFFE,BYTE_TO_INT(Crosstable[HeadAddr].NodeId) -33);
					ELSE
						CommErrTCPRTUL:=CommErrTCPRTUL AND ROL(16#FFFFFFFE,BYTE_TO_INT(Crosstable[HeadAddr].NodeId)-1 );
						k:=ROL(16#FFFFFFFE,BYTE_TO_INT(Crosstable[HeadAddr].NodeId)-1 );
						j:=BlackListTCPRTUL;
						j:=j AND k;
						BlackListTCPRTUL:=j;
					END_IF;
					IF CommErrTCPRTUH =0 AND CommErrTCPRTUl = 0 THEN
						TCPRTUComm_ERROR_WORD:=0;
					END_IF;
					IF BlackListTCPRTUH =0 AND BlackListTCPRTUL = 0 THEN
						TCPRTUBlackList_ERROR_WORD:=0;
					END_IF;

					TCPRTUListDevices[BYTE_TO_INT(Crosstable[HeadAddr].NodeId)].BlackListed:=0;
					TCPRTUListDevices[BYTE_TO_INT(Crosstable[HeadAddr].NodeId)].RetryCounter:=0;
				END_IF;
			ELSE
				TCPRTUListDevices[BYTE_TO_INT(Crosstable[HeadAddr].NodeId)].JumpRead:=TCPRTUListDevices[BYTE_TO_INT(Crosstable[HeadAddr].NodeId)].JumpRead-1;
				IF TCPRTUListDevices[BYTE_TO_INT(Crosstable[HeadAddr].NodeId)].JumpRead <= 0 THEN
					TCPRTUListDevices[BYTE_TO_INT(Crosstable[HeadAddr].NodeId)].BlackListed:=1;
					Retry:=TRUE;
				END_IF;
			END_IF;
		END_IF;
	END_IF;
END_IF;

END_PROGRAM
